FUNCTION WRITE_PROTECTED_UINT
VAR_INPUT
    Ptr : POINTER TO UINT;
    Value : UINT;
END_VAR

Ptr^ := Value;

END_FUNCTION

(* stored: Version 1.1.0.1, ProductVersion 3.1.4022.18
   POU WRITE_PROTECTED_UINT: Id {4b5114b2-1dc0-4e59-81df-bbfea3eeaaa0}, SpecialFunc None *)
